FUNCTION ASSEMBLE_LWORD_FROM_BOOLS (* this Function combines the 64 BOOLS to a LWORD *)
  (* Standard: 61499-1; Description: Copyright (c) 2024 HR Agrartechnik GmbH This program and the accompanying materials are made available under the terms of the Eclipse Public License 2.0 which is available at https://www.eclipse.org/legal/epl-2.0/ SPDX-License-Identifier: EPL-2.0 *)
  (* Version 3.0.1, 2026-09-29, Martin Jobst, fix ST package declaration *)
  (* Version 3.0, 2025-04-14, Patrick Aigner, changed package *)
  (* Version 1.1, 2024-07-28, Moritz Ortmeier, HR Agrartechnik, rename Function and change Input/Output Variables *)
  (* Version 1.0, 2024-02-22, Franz Höpfinger, HR Agrartechnik, initial Implementation *)
  PACKAGE eclipse4diac::utils::assembling;
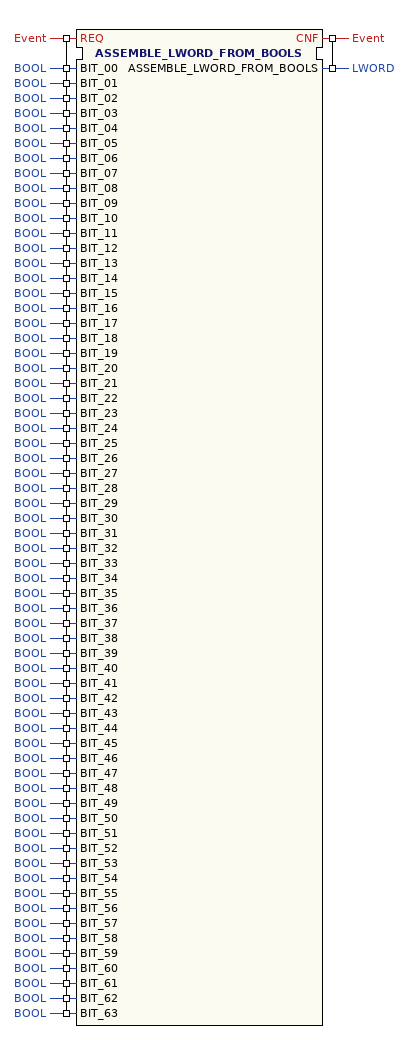
  EVENT_INPUT
    REQ WITH BIT_00, BIT_01, BIT_02, BIT_03, BIT_04, BIT_05, BIT_06, BIT_07, BIT_08, BIT_09, BIT_10, BIT_11, BIT_12, BIT_13, BIT_14, BIT_15, BIT_16, BIT_17, BIT_18, BIT_19, BIT_20, BIT_21, BIT_22, BIT_23, BIT_24, BIT_25, BIT_26, BIT_27, BIT_28, BIT_29, BIT_30, BIT_31, BIT_32, BIT_33, BIT_34, BIT_35, BIT_36, BIT_37, BIT_38, BIT_39, BIT_40, BIT_41, BIT_42, BIT_43, BIT_44, BIT_45, BIT_46, BIT_47, BIT_48, BIT_49, BIT_50, BIT_51, BIT_52, BIT_53, BIT_54, BIT_55, BIT_56, BIT_57, BIT_58, BIT_59, BIT_60, BIT_61, BIT_62, BIT_63;
  END_EVENT
  EVENT_OUTPUT
    CNF WITH ASSEMBLE_LWORD_FROM_BOOLS;
  END_EVENT
  VAR_INPUT
    BIT_00 : BOOL;
    BIT_01 : BOOL;
    BIT_02 : BOOL;
    BIT_03 : BOOL;
    BIT_04 : BOOL;
    BIT_05 : BOOL;
    BIT_06 : BOOL;
    BIT_07 : BOOL;
    BIT_08 : BOOL;
    BIT_09 : BOOL;
    BIT_10 : BOOL;
    BIT_11 : BOOL;
    BIT_12 : BOOL;
    BIT_13 : BOOL;
    BIT_14 : BOOL;
    BIT_15 : BOOL;
    BIT_16 : BOOL;
    BIT_17 : BOOL;
    BIT_18 : BOOL;
    BIT_19 : BOOL;
    BIT_20 : BOOL;
    BIT_21 : BOOL;
    BIT_22 : BOOL;
    BIT_23 : BOOL;
    BIT_24 : BOOL;
    BIT_25 : BOOL;
    BIT_26 : BOOL;
    BIT_27 : BOOL;
    BIT_28 : BOOL;
    BIT_29 : BOOL;
    BIT_30 : BOOL;
    BIT_31 : BOOL;
    BIT_32 : BOOL;
    BIT_33 : BOOL;
    BIT_34 : BOOL;
    BIT_35 : BOOL;
    BIT_36 : BOOL;
    BIT_37 : BOOL;
    BIT_38 : BOOL;
    BIT_39 : BOOL;
    BIT_40 : BOOL;
    BIT_41 : BOOL;
    BIT_42 : BOOL;
    BIT_43 : BOOL;
    BIT_44 : BOOL;
    BIT_45 : BOOL;
    BIT_46 : BOOL;
    BIT_47 : BOOL;
    BIT_48 : BOOL;
    BIT_49 : BOOL;
    BIT_50 : BOOL;
    BIT_51 : BOOL;
    BIT_52 : BOOL;
    BIT_53 : BOOL;
    BIT_54 : BOOL;
    BIT_55 : BOOL;
    BIT_56 : BOOL;
    BIT_57 : BOOL;
    BIT_58 : BOOL;
    BIT_59 : BOOL;
    BIT_60 : BOOL;
    BIT_61 : BOOL;
    BIT_62 : BOOL;
    BIT_63 : BOOL;
  END_VAR
  VAR_OUTPUT
    ASSEMBLE_LWORD_FROM_BOOLS : LWORD;
  END_VAR
  BODY IN ST:
PACKAGE eclipse4diac::utils::assembling;

(* this Function combines the 64 BOOLS to a LWORD *)
FUNCTION ASSEMBLE_LWORD_FROM_BOOLS : LWORD

VAR_INPUT
	BIT_00 : BOOL;
	BIT_01 : BOOL;
	BIT_02 : BOOL;
	BIT_03 : BOOL;
	BIT_04 : BOOL;
	BIT_05 : BOOL;
	BIT_06 : BOOL;
	BIT_07 : BOOL;
	BIT_08 : BOOL;
	BIT_09 : BOOL;
	BIT_10 : BOOL;
	BIT_11 : BOOL;
	BIT_12 : BOOL;
	BIT_13 : BOOL;
	BIT_14 : BOOL;
	BIT_15 : BOOL;
	BIT_16 : BOOL;
	BIT_17 : BOOL;
	BIT_18 : BOOL;
	BIT_19 : BOOL;
	BIT_20 : BOOL;
	BIT_21 : BOOL;
	BIT_22 : BOOL;
	BIT_23 : BOOL;
	BIT_24 : BOOL;
	BIT_25 : BOOL;
	BIT_26 : BOOL;
	BIT_27 : BOOL;
	BIT_28 : BOOL;
	BIT_29 : BOOL;
	BIT_30 : BOOL;
	BIT_31 : BOOL;
	BIT_32 : BOOL;
	BIT_33 : BOOL;
	BIT_34 : BOOL;
	BIT_35 : BOOL;
	BIT_36 : BOOL;
	BIT_37 : BOOL;
	BIT_38 : BOOL;
	BIT_39 : BOOL;
	BIT_40 : BOOL;
	BIT_41 : BOOL;
	BIT_42 : BOOL;
	BIT_43 : BOOL;
	BIT_44 : BOOL;
	BIT_45 : BOOL;
	BIT_46 : BOOL;
	BIT_47 : BOOL;
	BIT_48 : BOOL;
	BIT_49 : BOOL;
	BIT_50 : BOOL;
	BIT_51 : BOOL;
	BIT_52 : BOOL;
	BIT_53 : BOOL;
	BIT_54 : BOOL;
	BIT_55 : BOOL;
	BIT_56 : BOOL;
	BIT_57 : BOOL;
	BIT_58 : BOOL;
	BIT_59 : BOOL;
	BIT_60 : BOOL;
	BIT_61 : BOOL;
	BIT_62 : BOOL;
	BIT_63 : BOOL;
END_VAR

ASSEMBLE_LWORD_FROM_BOOLS.%X0 := BIT_00;
ASSEMBLE_LWORD_FROM_BOOLS.%X1 := BIT_01;
ASSEMBLE_LWORD_FROM_BOOLS.%X2 := BIT_02;
ASSEMBLE_LWORD_FROM_BOOLS.%X3 := BIT_03;
ASSEMBLE_LWORD_FROM_BOOLS.%X4 := BIT_04;
ASSEMBLE_LWORD_FROM_BOOLS.%X5 := BIT_05;
ASSEMBLE_LWORD_FROM_BOOLS.%X6 := BIT_06;
ASSEMBLE_LWORD_FROM_BOOLS.%X7 := BIT_07;
ASSEMBLE_LWORD_FROM_BOOLS.%X8 := BIT_08;
ASSEMBLE_LWORD_FROM_BOOLS.%X9 := BIT_09;
ASSEMBLE_LWORD_FROM_BOOLS.%X10 := BIT_10;
ASSEMBLE_LWORD_FROM_BOOLS.%X11 := BIT_11;
ASSEMBLE_LWORD_FROM_BOOLS.%X12 := BIT_12;
ASSEMBLE_LWORD_FROM_BOOLS.%X13 := BIT_13;
ASSEMBLE_LWORD_FROM_BOOLS.%X14 := BIT_14;
ASSEMBLE_LWORD_FROM_BOOLS.%X15 := BIT_15;
ASSEMBLE_LWORD_FROM_BOOLS.%X16 := BIT_16;
ASSEMBLE_LWORD_FROM_BOOLS.%X17 := BIT_17;
ASSEMBLE_LWORD_FROM_BOOLS.%X18 := BIT_18;
ASSEMBLE_LWORD_FROM_BOOLS.%X19 := BIT_19;
ASSEMBLE_LWORD_FROM_BOOLS.%X20 := BIT_20;
ASSEMBLE_LWORD_FROM_BOOLS.%X21 := BIT_21;
ASSEMBLE_LWORD_FROM_BOOLS.%X22 := BIT_22;
ASSEMBLE_LWORD_FROM_BOOLS.%X23 := BIT_23;
ASSEMBLE_LWORD_FROM_BOOLS.%X24 := BIT_24;
ASSEMBLE_LWORD_FROM_BOOLS.%X25 := BIT_25;
ASSEMBLE_LWORD_FROM_BOOLS.%X26 := BIT_26;
ASSEMBLE_LWORD_FROM_BOOLS.%X27 := BIT_27;
ASSEMBLE_LWORD_FROM_BOOLS.%X28 := BIT_28;
ASSEMBLE_LWORD_FROM_BOOLS.%X29 := BIT_29;
ASSEMBLE_LWORD_FROM_BOOLS.%X30 := BIT_30;
ASSEMBLE_LWORD_FROM_BOOLS.%X31 := BIT_31;
ASSEMBLE_LWORD_FROM_BOOLS.%X32 := BIT_32;
ASSEMBLE_LWORD_FROM_BOOLS.%X33 := BIT_33;
ASSEMBLE_LWORD_FROM_BOOLS.%X34 := BIT_34;
ASSEMBLE_LWORD_FROM_BOOLS.%X35 := BIT_35;
ASSEMBLE_LWORD_FROM_BOOLS.%X36 := BIT_36;
ASSEMBLE_LWORD_FROM_BOOLS.%X37 := BIT_37;
ASSEMBLE_LWORD_FROM_BOOLS.%X38 := BIT_38;
ASSEMBLE_LWORD_FROM_BOOLS.%X39 := BIT_39;
ASSEMBLE_LWORD_FROM_BOOLS.%X40 := BIT_40;
ASSEMBLE_LWORD_FROM_BOOLS.%X41 := BIT_41;
ASSEMBLE_LWORD_FROM_BOOLS.%X42 := BIT_42;
ASSEMBLE_LWORD_FROM_BOOLS.%X43 := BIT_43;
ASSEMBLE_LWORD_FROM_BOOLS.%X44 := BIT_44;
ASSEMBLE_LWORD_FROM_BOOLS.%X45 := BIT_45;
ASSEMBLE_LWORD_FROM_BOOLS.%X46 := BIT_46;
ASSEMBLE_LWORD_FROM_BOOLS.%X47 := BIT_47;
ASSEMBLE_LWORD_FROM_BOOLS.%X48 := BIT_48;
ASSEMBLE_LWORD_FROM_BOOLS.%X49 := BIT_49;
ASSEMBLE_LWORD_FROM_BOOLS.%X50 := BIT_50;
ASSEMBLE_LWORD_FROM_BOOLS.%X51 := BIT_51;
ASSEMBLE_LWORD_FROM_BOOLS.%X52 := BIT_52;
ASSEMBLE_LWORD_FROM_BOOLS.%X53 := BIT_53;
ASSEMBLE_LWORD_FROM_BOOLS.%X54 := BIT_54;
ASSEMBLE_LWORD_FROM_BOOLS.%X55 := BIT_55;
ASSEMBLE_LWORD_FROM_BOOLS.%X56 := BIT_56;
ASSEMBLE_LWORD_FROM_BOOLS.%X57 := BIT_57;
ASSEMBLE_LWORD_FROM_BOOLS.%X58 := BIT_58;
ASSEMBLE_LWORD_FROM_BOOLS.%X59 := BIT_59;
ASSEMBLE_LWORD_FROM_BOOLS.%X60 := BIT_60;
ASSEMBLE_LWORD_FROM_BOOLS.%X61 := BIT_61;
ASSEMBLE_LWORD_FROM_BOOLS.%X62 := BIT_62;
ASSEMBLE_LWORD_FROM_BOOLS.%X63 := BIT_63;
END_FUNCTION
  END_BODY
END_FUNCTION
